(* PLC project Tc2_Utilities.FB_GetSystemId Demo, tc3-libraries-kb TwinCAT 3.1 *)
(* stored: creationDateTime 2026-05-11T00:00:00, modificationDateTime 2026-05-11T00:00:00 *)

PROGRAM P_Demo_FB_GetSystemId
  VAR
    fbFB_GetSystemId : FB_GetSystemId;  (* FB_GetSystemId 实例 *)
    bRead : BOOL := FALSE;
    systemId : GUID;  (* 本机 SystemID *)
    bBusy_ : BOOL;
    bErrFlag : BOOL;
    nErrCode : UDINT;
  END_VAR

// =============================================================================
// 场景：License POU 启动时读一次 SystemID 做校验。
// 价值：标准 License 绑定锚点。
// 验证：改 bRead := TRUE，观察 systemId 装载 16 字节 GUID（非全 0）。
// 验证步骤：
//   1. 右键 PLC 项目 → Import PLCopenXML → 选本文件
//   2. 引用 Tc2_Utilities（References → Add library）
//   3. 编译 → 登录 → 运行；按上方『验证』行的指示在线写值观察
// =============================================================================

fbFB_GetSystemId(
    bExecute := bRead,
    tTimeout := DEFAULT_ADS_TIMEOUT,
    systemId => systemId,
    bBusy => bBusy_,
    bErr => bErrFlag,
    nErrId => nErrCode
);
END_PROGRAM
